TYPE ST_Parameters_MR :
STRUCT
	methodName			: STRING(100);
	methodRevision		: STRING(100);
	methodCreatedBy		: STRING(100);
	methodCreatedOn		: STRING(100);
	solvent_R1			: STRING(100);
	solvent_R2			: STRING(100);
	solvent_W1			: STRING(100);
	solvent_W2			: STRING(100);
	time_R1				: STRING(100);
	time_R2				: STRING(100);
	time_W1				: STRING(100);
	time_W2				: STRING(100);	
	velocity_R1			: STRING(100);
	velocity_R2			: STRING(100);
	velocity_W1			: STRING(100);
	velocity_W2			: STRING(100);
	soakTime			: STRING(100);
	agitate_1_Time		: STRING(100);
	agitate_2_Time		: STRING(100);
	vialsToFill			: STRING(100);
	vialPrimeVol		: STRING(100);
	vial_1_FillVol		: STRING(100);
	vial_2_4_FillVol	: STRING(100);
	airDryTime			: STRING(100);
	methodID			: INT;
	methodStatus		: STRING(100);
	
END_STRUCT
END_TYPE

(* stored: Version 1.1.0.1, ProductVersion 3.1.4024.15
   DUT ST_Parameters_MR: Id {f829ad56-d934-44b7-9430-3c29a09c0980} *)
